{attribute 'GeneratedUsingTerminal: EL1918-0000-0016'}
{attribute addProperty BoxType "EL1918-0000-0016"}
{attribute addProperty Id "FSOEAT %Q*FSOE_3054F84313"}
{attribute addProperty CRC "1496771782"}
{attribute addProperty Size "13"}
TYPE FSoE_Outputs_5936ECC6 EXTENDS OutputBase_10CEE7DE :
STRUCT
	{attribute addProperty Name "FSOE"}
	FSOE AT %Q* : FSOE_3054F843;
END_STRUCT
END_TYPE

(* stored: Version 1.2.0.0, ProductVersion 3.1.4024.9
   DUT FSoE_Outputs_5936ECC6: Id {709ddb98-c6b5-4354-9e86-e2eba4d20bf8} *)
